{attribute addProperty BoxType "APS4322-7000-0017"}
{attribute addProperty Id "StatusWordAT %I*UINT16217Current_D_0X0AT %I*INT1622Current_D_0X1AT %I*INT1623Current_D_0X2AT %I*INT1624Current_D_0Y0AT %I*INT1625Current_D_0Y1AT %I*INT1626Current_D_0Y2AT %I*INT1627Current_D_1X0AT %I*INT1628Current_D_1X1AT %I*INT1629Current_D_1X2AT %I*INT16210Current_D_1Y0AT %I*INT16211Current_D_1Y1AT %I*INT16212Current_D_1Y2AT %I*INT16213Current_D_2X0AT %I*INT16214Current_D_2X1AT %I*INT16215Current_D_2X2AT %I*INT16216Current_D_2Y0AT %I*INT16217Current_D_2Y1AT %I*INT16218Current_D_2Y2AT %I*INT16219Current_D_3X0AT %I*INT16220Current_D_3X1AT %I*INT16221Current_D_3X2AT %I*INT16222Current_D_3Y0AT %I*INT16223Current_D_3Y1AT %I*INT16224Current_D_3Y2AT %I*INT16225Current_Q_0X0AT %I*INT16226Current_Q_0X1AT %I*INT16227Current_Q_0X2AT %I*INT16228Current_Q_0Y0AT %I*INT16229Current_Q_0Y1AT %I*INT16230Current_Q_0Y2AT %I*INT16231Current_Q_1X0AT %I*INT16232Current_Q_1X1AT %I*INT16233Current_Q_1X2AT %I*INT16234Current_Q_1Y0AT %I*INT16235Current_Q_1Y1AT %I*INT16236Current_Q_1Y2AT %I*INT16237Current_Q_2X0AT %I*INT16238Current_Q_2X1AT %I*INT16239Current_Q_2X2AT %I*INT16240Current_Q_2Y0AT %I*INT16241Current_Q_2Y1AT %I*INT16242Current_Q_2Y2AT %I*INT16243Current_Q_3X0AT %I*INT16244Current_Q_3X1AT %I*INT16245Current_Q_3X2AT %I*INT16246Current_Q_3Y0AT %I*INT16247Current_Q_3Y1AT %I*INT16248Current_Q_3Y2AT %I*INT16249"}
{attribute addProperty CRC "850592125"}
{attribute addProperty SizeInBites "784"}
{attribute addProperty SizeInBytes "98"}
TYPE APS_Inputs_32B3017D :
STRUCT
	{attribute addProperty Name "StatusWord"}
	StatusWord AT %I* : UINT;
	{attribute addProperty Name "Current_D_0X0"}
	Current_D_0X0 AT %I* : INT;
	{attribute addProperty Name "Current_D_0X1"}
	Current_D_0X1 AT %I* : INT;
	{attribute addProperty Name "Current_D_0X2"}
	Current_D_0X2 AT %I* : INT;
	{attribute addProperty Name "Current_D_0Y0"}
	Current_D_0Y0 AT %I* : INT;
	{attribute addProperty Name "Current_D_0Y1"}
	Current_D_0Y1 AT %I* : INT;
	{attribute addProperty Name "Current_D_0Y2"}
	Current_D_0Y2 AT %I* : INT;
	{attribute addProperty Name "Current_D_1X0"}
	Current_D_1X0 AT %I* : INT;
	{attribute addProperty Name "Current_D_1X1"}
	Current_D_1X1 AT %I* : INT;
	{attribute addProperty Name "Current_D_1X2"}
	Current_D_1X2 AT %I* : INT;
	{attribute addProperty Name "Current_D_1Y0"}
	Current_D_1Y0 AT %I* : INT;
	{attribute addProperty Name "Current_D_1Y1"}
	Current_D_1Y1 AT %I* : INT;
	{attribute addProperty Name "Current_D_1Y2"}
	Current_D_1Y2 AT %I* : INT;
	{attribute addProperty Name "Current_D_2X0"}
	Current_D_2X0 AT %I* : INT;
	{attribute addProperty Name "Current_D_2X1"}
	Current_D_2X1 AT %I* : INT;
	{attribute addProperty Name "Current_D_2X2"}
	Current_D_2X2 AT %I* : INT;
	{attribute addProperty Name "Current_D_2Y0"}
	Current_D_2Y0 AT %I* : INT;
	{attribute addProperty Name "Current_D_2Y1"}
	Current_D_2Y1 AT %I* : INT;
	{attribute addProperty Name "Current_D_2Y2"}
	Current_D_2Y2 AT %I* : INT;
	{attribute addProperty Name "Current_D_3X0"}
	Current_D_3X0 AT %I* : INT;
	{attribute addProperty Name "Current_D_3X1"}
	Current_D_3X1 AT %I* : INT;
	{attribute addProperty Name "Current_D_3X2"}
	Current_D_3X2 AT %I* : INT;
	{attribute addProperty Name "Current_D_3Y0"}
	Current_D_3Y0 AT %I* : INT;
	{attribute addProperty Name "Current_D_3Y1"}
	Current_D_3Y1 AT %I* : INT;
	{attribute addProperty Name "Current_D_3Y2"}
	Current_D_3Y2 AT %I* : INT;
	{attribute addProperty Name "Current_Q_0X0"}
	Current_Q_0X0 AT %I* : INT;
	{attribute addProperty Name "Current_Q_0X1"}
	Current_Q_0X1 AT %I* : INT;
	{attribute addProperty Name "Current_Q_0X2"}
	Current_Q_0X2 AT %I* : INT;
	{attribute addProperty Name "Current_Q_0Y0"}
	Current_Q_0Y0 AT %I* : INT;
	{attribute addProperty Name "Current_Q_0Y1"}
	Current_Q_0Y1 AT %I* : INT;
	{attribute addProperty Name "Current_Q_0Y2"}
	Current_Q_0Y2 AT %I* : INT;
	{attribute addProperty Name "Current_Q_1X0"}
	Current_Q_1X0 AT %I* : INT;
	{attribute addProperty Name "Current_Q_1X1"}
	Current_Q_1X1 AT %I* : INT;
	{attribute addProperty Name "Current_Q_1X2"}
	Current_Q_1X2 AT %I* : INT;
	{attribute addProperty Name "Current_Q_1Y0"}
	Current_Q_1Y0 AT %I* : INT;
	{attribute addProperty Name "Current_Q_1Y1"}
	Current_Q_1Y1 AT %I* : INT;
	{attribute addProperty Name "Current_Q_1Y2"}
	Current_Q_1Y2 AT %I* : INT;
	{attribute addProperty Name "Current_Q_2X0"}
	Current_Q_2X0 AT %I* : INT;
	{attribute addProperty Name "Current_Q_2X1"}
	Current_Q_2X1 AT %I* : INT;
	{attribute addProperty Name "Current_Q_2X2"}
	Current_Q_2X2 AT %I* : INT;
	{attribute addProperty Name "Current_Q_2Y0"}
	Current_Q_2Y0 AT %I* : INT;
	{attribute addProperty Name "Current_Q_2Y1"}
	Current_Q_2Y1 AT %I* : INT;
	{attribute addProperty Name "Current_Q_2Y2"}
	Current_Q_2Y2 AT %I* : INT;
	{attribute addProperty Name "Current_Q_3X0"}
	Current_Q_3X0 AT %I* : INT;
	{attribute addProperty Name "Current_Q_3X1"}
	Current_Q_3X1 AT %I* : INT;
	{attribute addProperty Name "Current_Q_3X2"}
	Current_Q_3X2 AT %I* : INT;
	{attribute addProperty Name "Current_Q_3Y0"}
	Current_Q_3Y0 AT %I* : INT;
	{attribute addProperty Name "Current_Q_3Y1"}
	Current_Q_3Y1 AT %I* : INT;
	{attribute addProperty Name "Current_Q_3Y2"}
	Current_Q_3Y2 AT %I* : INT;
END_STRUCT
END_TYPE

(* stored: Version 1.2.0.0, ProductVersion 3.1.4024.9
   DUT APS_Inputs_32B3017D: Id {99ea5021-7220-4499-a232-f3a3844c44ba} *)
